KUKA KRL program: Milling_7_2.src

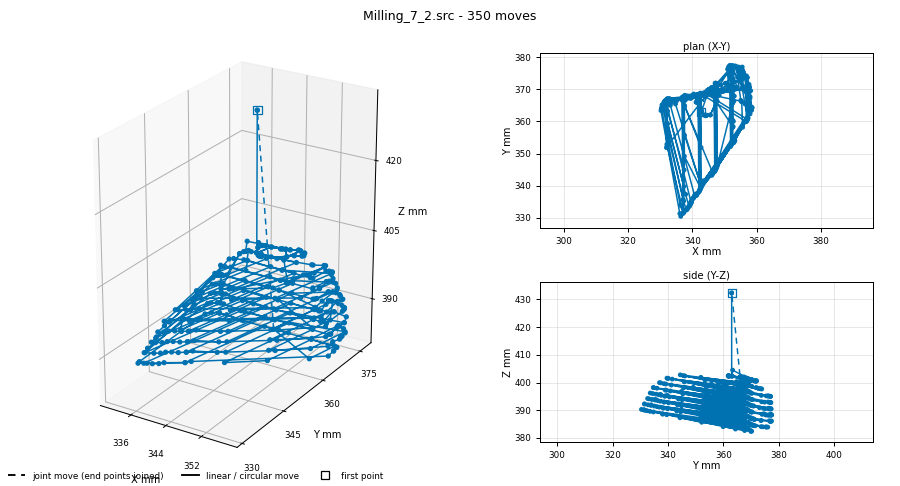
[picture p0: tool path of Milling_7_2.src, 350 of 352 moves have a stored position in this frame; points joined in program order, loops and branches not executed]
&ACCESS RVP
&REL 1
&PARAM TEMPLATE = C:\KRC\Roboter\Template\vorgabe
&PARAM EDITMASK = *
DEF Milling_7_2 ( )


;FOLD INI
;FOLD BASISTECH INI
GLOBAL INTERRUPT DECL 3 WHEN $STOPMESS==TRUE DO IR_STOPM ( )
INTERRUPT ON 3
BAS (#INITMOV,0 )
;ENDFOLD (BASISTECH INI)
;ENDFOLD (INI)

;FOLD STARTPOSITION - BASE IS 0, TOOL IS 5, SPEED IS 15%, POSITION IS A1 5,A2 -90,A3 100,A4 5,A5 -10,A6 -5,E1 0,E2 0,E3 0,E4 0
$BWDSTART = FALSE
PDAT_ACT = {VEL 15,ACC 100,APO_DIST 50}
FDAT_ACT = {TOOL_NO 5,BASE_NO 0,IPO_FRAME #BASE}
BAS (#PTP_PARAMS,15)
PTP  {A1 5,A2 -90,A3 100,A4 5,A5 -10,A6 -5,E1 0,E2 0,E3 0,E4 0}
;ENDFOLD

;FOLD LIN SPEED IS 0.1 m/sec, INTERPOLATION SETTINGS IN FOLD
$VEL.CP=0.1
$ADVANCE=3
;ENDFOLD

BAS(#VEL_PTP,2)
PTP {X 342.707, Y 362.992, Z 432.358, A -116.805, B 80.034, C -131.472, E1 0, E2 0, E3 0, E4 0, S 'B010'}
$VEL.CP=0.012
LIN {X 342.707, Y 362.992, Z 402.358, A -116.805, B 80.034, C -131.472, E1 0, E2 0, E3 0, E4 0}
LIN {X 342.661, Y 368.658, Z 401.473, A -116.805, B 80.034, C -131.472, E1 0, E2 0, E3 0, E4 0}
LIN {X 347.621, Y 371.786, Z 400.589, A -116.805, B 80.034, C -131.472, E1 0, E2 0, E3 0, E4 0}
LIN {X 347.667, Y 366.252, Z 401.453, A -116.805, B 80.034, C -131.472, E1 0, E2 0, E3 0, E4 0}
LIN {X 345.179, Y 369.984, Z 401.065, A -116.805, B 80.034, C -131.472, E1 0, E2 0, E3 0, E4 0}
LIN {X 345.924, Y 370.498, Z 400.926, A -116.805, B 80.034, C -131.472, E1 0, E2 0, E3 0, E4 0}
LIN {X 347.063, Y 371.85, Z 400.623, A -116.805, B 80.034, C -131.472, E1 0, E2 0, E3 0, E4 0}
LIN {X 347.223, Y 371.899, Z 400.603, A -116.805, B 80.034, C -131.472, E1 0, E2 0, E3 0, E4 0}
LIN {X 348.776, Y 371.334, Z 400.569, A -116.805, B 80.034, C -131.472, E1 0, E2 0, E3 0, E4 0}
LIN {X 349.45, Y 369.842, Z 400.749, A -116.805, B 80.034, C -131.472, E1 0, E2 0, E3 0, E4 0}
LIN {X 349.322, Y 369.366, Z 400.834, A -116.805, B 80.034, C -131.472, E1 0, E2 0, E3 0, E4 0}
LIN {X 348.261, Y 368.158, Z 401.107, A -116.805, B 80.034, C -131.472, E1 0, E2 0, E3 0, E4 0}
LIN {X 345.56, Y 361.988, Z 402.289, A -116.805, B 80.034, C -131.472, E1 0, E2 0, E3 0, E4 0}
LIN {X 344.437, Y 361.921, Z 402.389, A -116.805, B 80.034, C -131.472, E1 0, E2 0, E3 0, E4 0}
LIN {X 344.141, Y 361.749, Z 402.439, A -116.805, B 80.034, C -131.472, E1 0, E2 0, E3 0, E4 0}
LIN {X 343.696, Y 361.979, Z 402.438, A -116.805, B 80.034, C -131.472, E1 0, E2 0, E3 0, E4 0}
LIN {X 342.553, Y 363.151, Z 402.345, A -116.805, B 80.034, C -131.472, E1 0, E2 0, E3 0, E4 0}
LIN {X 341.15, Y 365.964, Z 402.015, A -116.805, B 80.034, C -131.472, E1 0, E2 0, E3 0, E4 0}
LIN {X 341.012, Y 367.77, Z 401.743, A -116.805, B 80.034, C -131.472, E1 0, E2 0, E3 0, E4 0}
LIN {X 341.478, Y 368.328, Z 401.618, A -116.805, B 80.034, C -131.472, E1 0, E2 0, E3 0, E4 0}
LIN {X 344.42, Y 369.322, Z 401.229, A -116.805, B 80.034, C -131.472, E1 0, E2 0, E3 0, E4 0}
LIN {X 344.649, Y 369.619, Z 401.165, A -116.805, B 80.034, C -131.472, E1 0, E2 0, E3 0, E4 0}
LIN {X 345.179, Y 369.984, Z 401.065, A -116.805, B 80.034, C -131.472, E1 0, E2 0, E3 0, E4 0}
LIN {X 342.877, Y 363.328, Z 404.499, A -116.805, B 80.034, C -131.472, E1 0, E2 0, E3 0, E4 0}
LIN {X 342.707, Y 362.992, Z 402.358, A -116.805, B 80.034, C -131.472, E1 0, E2 0, E3 0, E4 0}
LIN {X 342.661, Y 368.658, Z 401.473, A -116.805, B 80.034, C -131.472, E1 0, E2 0, E3 0, E4 0}
LIN {X 347.621, Y 371.786, Z 400.589, A -116.805, B 80.034, C -131.472, E1 0, E2 0, E3 0, E4 0}
LIN {X 347.667, Y 366.252, Z 401.453, A -116.805, B 80.034, C -131.472, E1 0, E2 0, E3 0, E4 0}
LIN {X 345.179, Y 369.984, Z 401.065, A -116.805, B 80.034, C -131.472, E1 0, E2 0, E3 0, E4 0}
LIN {X 345.924, Y 370.498, Z 400.926, A -116.805, B 80.034, C -131.472, E1 0, E2 0, E3 0, E4 0}
LIN {X 347.063, Y 371.85, Z 400.623, A -116.805, B 80.034, C -131.472, E1 0, E2 0, E3 0, E4 0}
LIN {X 347.223, Y 371.899, Z 400.603, A -116.805, B 80.034, C -131.472, E1 0, E2 0, E3 0, E4 0}
LIN {X 348.776, Y 371.334, Z 400.569, A -116.805, B 80.034, C -131.472, E1 0, E2 0, E3 0, E4 0}
LIN {X 349.45, Y 369.842, Z 400.749, A -116.805, B 80.034, C -131.472, E1 0, E2 0, E3 0, E4 0}
LIN {X 349.322, Y 369.366, Z 400.834, A -116.805, B 80.034, C -131.472, E1 0, E2 0, E3 0, E4 0}
LIN {X 348.261, Y 368.158, Z 401.107, A -116.805, B 80.034, C -131.472, E1 0, E2 0, E3 0, E4 0}
LIN {X 345.56, Y 361.988, Z 402.289, A -116.805, B 80.034, C -131.472, E1 0, E2 0, E3 0, E4 0}
LIN {X 344.437, Y 361.921, Z 402.389, A -116.805, B 80.034, C -131.472, E1 0, E2 0, E3 0, E4 0}
LIN {X 344.141, Y 361.749, Z 402.439, A -116.805, B 80.034, C -131.472, E1 0, E2 0, E3 0, E4 0}
LIN {X 343.696, Y 361.979, Z 402.438, A -116.805, B 80.034, C -131.472, E1 0, E2 0, E3 0, E4 0}
LIN {X 342.553, Y 363.151, Z 402.345, A -116.805, B 80.034, C -131.472, E1 0, E2 0, E3 0, E4 0}
LIN {X 341.15, Y 365.964, Z 402.015, A -116.805, B 80.034, C -131.472, E1 0, E2 0, E3 0, E4 0}
LIN {X 341.012, Y 367.77, Z 401.743, A -116.805, B 80.034, C -131.472, E1 0, E2 0, E3 0, E4 0}
LIN {X 341.478, Y 368.328, Z 401.618, A -116.805, B 80.034, C -131.472, E1 0, E2 0, E3 0, E4 0}
LIN {X 344.42, Y 369.322, Z 401.229, A -116.805, B 80.034, C -131.472, E1 0, E2 0, E3 0, E4 0}
LIN {X 344.649, Y 369.619, Z 401.165, A -116.805, B 80.034, C -131.472, E1 0, E2 0, E3 0, E4 0}
LIN {X 345.179, Y 369.984, Z 401.065, A -116.805, B 80.034, C -131.472, E1 0, E2 0, E3 0, E4 0}
LIN {X 337.743, Y 367.407, Z 402.059, A -116.805, B 80.034, C -131.472, E1 0, E2 0, E3 0, E4 0}
LIN {X 337.573, Y 367.071, Z 399.918, A -116.805, B 80.034, C -131.472, E1 0, E2 0, E3 0, E4 0}
LIN {X 337.592, Y 364.763, Z 400.278, A -116.805, B 80.034, C -131.472, E1 0, E2 0, E3 0, E4 0}
LIN {X 342.685, Y 351.876, Z 401.896, A -116.805, B 80.034, C -131.472, E1 0, E2 0, E3 0, E4 0}
LIN {X 342.545, Y 368.751, Z 399.26, A -116.805, B 80.034, C -131.472, E1 0, E2 0, E3 0, E4 0}
LIN {X 347.519, Y 370.271, Z 398.628, A -116.805, B 80.034, C -131.472, E1 0, E2 0, E3 0, E4 0}
LIN {X 347.718, Y 346.142, Z 402.396, A -116.805, B 80.034, C -131.472, E1 0, E2 0, E3 0, E4 0}
LIN {X 352.543, Y 365.664, Z 398.952, A -116.805, B 80.034, C -131.472, E1 0, E2 0, E3 0, E4 0}
LIN {X 352.483, Y 372.939, Z 397.816, A -116.805, B 80.034, C -131.472, E1 0, E2 0, E3 0, E4 0}
LIN {X 352.587, Y 360.294, Z 399.791, A -116.805, B 80.034, C -131.472, E1 0, E2 0, E3 0, E4 0}
LIN {X 352.604, Y 358.316, Z 400.1, A -116.805, B 80.034, C -131.472, E1 0, E2 0, E3 0, E4 0}
LIN {X 345.127, Y 369.414, Z 398.952, A -116.805, B 80.034, C -131.472, E1 0, E2 0, E3 0, E4 0}
LIN {X 350.17, Y 371.833, Z 398.173, A -116.805, B 80.034, C -131.472, E1 0, E2 0, E3 0, E4 0}
LIN {X 350.43, Y 371.898, Z 398.142, A -116.805, B 80.034, C -131.472, E1 0, E2 0, E3 0, E4 0}
LIN {X 351.948, Y 373.669, Z 397.744, A -116.805, B 80.034, C -131.472, E1 0, E2 0, E3 0, E4 0}
LIN {X 352.209, Y 373.838, Z 397.697, A -116.805, B 80.034, C -131.472, E1 0, E2 0, E3 0, E4 0}
LIN {X 352.325, Y 373.23, Z 397.783, A -116.805, B 80.034, C -131.472, E1 0, E2 0, E3 0, E4 0}
LIN {X 352.575, Y 372.77, Z 397.835, A -116.805, B 80.034, C -131.472, E1 0, E2 0, E3 0, E4 0}
LIN {X 353.028, Y 367.871, Z 398.567, A -116.805, B 80.034, C -131.472, E1 0, E2 0, E3 0, E4 0}
LIN {X 352.901, Y 366.299, Z 398.824, A -116.805, B 80.034, C -131.472, E1 0, E2 0, E3 0, E4 0}
LIN {X 352.206, Y 365.066, Z 399.072, A -116.805, B 80.034, C -131.472, E1 0, E2 0, E3 0, E4 0}
LIN {X 352.083, Y 361.375, Z 399.661, A -116.805, B 80.034, C -131.472, E1 0, E2 0, E3 0, E4 0}
LIN {X 352.727, Y 359.98, Z 399.829, A -116.805, B 80.034, C -131.472, E1 0, E2 0, E3 0, E4 0}
LIN {X 352.636, Y 358.39, Z 400.085, A -116.805, B 80.034, C -131.472, E1 0, E2 0, E3 0, E4 0}
LIN {X 352.49, Y 358.055, Z 400.15, A -116.805, B 80.034, C -131.472, E1 0, E2 0, E3 0, E4 0}
LIN {X 352.27, Y 353.357, Z 400.904, A -116.805, B 80.034, C -131.472, E1 0, E2 0, E3 0, E4 0}
LIN {X 347.282, Y 345.532, Z 402.526, A -116.805, B 80.034, C -131.472, E1 0, E2 0, E3 0, E4 0}
LIN {X 346.146, Y 344.436, Z 402.788, A -116.805, B 80.034, C -131.472, E1 0, E2 0, E3 0, E4 0}
LIN {X 337.557, Y 364.832, Z 400.27, A -116.805, B 80.034, C -131.472, E1 0, E2 0, E3 0, E4 0}
LIN {X 337.427, Y 366.588, Z 400.005, A -116.805, B 80.034, C -131.472, E1 0, E2 0, E3 0, E4 0}
LIN {X 337.628, Y 367.255, Z 399.884, A -116.805, B 80.034, C -131.472, E1 0, E2 0, E3 0, E4 0}
LIN {X 338.367, Y 367.942, Z 399.718, A -116.805, B 80.034, C -131.472, E1 0, E2 0, E3 0, E4 0}
LIN {X 340.366, Y 368.526, Z 399.468, A -116.805, B 80.034, C -131.472, E1 0, E2 0, E3 0, E4 0}
LIN {X 343.878, Y 368.815, Z 399.145, A -116.805, B 80.034, C -131.472, E1 0, E2 0, E3 0, E4 0}
LIN {X 345.127, Y 369.414, Z 398.952, A -116.805, B 80.034, C -131.472, E1 0, E2 0, E3 0, E4 0}
LIN {X 337.622, Y 368.124, Z 399.749, A -116.805, B 80.034, C -131.472, E1 0, E2 0, E3 0, E4 0}
LIN {X 337.452, Y 367.788, Z 397.607, A -116.805, B 80.034, C -131.472, E1 0, E2 0, E3 0, E4 0}
LIN {X 337.553, Y 355.652, Z 399.503, A -116.805, B 80.034, C -131.472, E1 0, E2 0, E3 0, E4 0}
LIN {X 342.668, Y 340.052, Z 401.544, A -116.805, B 80.034, C -131.472, E1 0, E2 0, E3 0, E4 0}
LIN {X 342.43, Y 368.782, Z 397.057, A -116.805, B 80.034, C -131.472, E1 0, E2 0, E3 0, E4 0}
LIN {X 347.41, Y 369.598, Z 396.535, A -116.805, B 80.034, C -131.472, E1 0, E2 0, E3 0, E4 0}
LIN {X 347.606, Y 345.887, Z 400.238, A -116.805, B 80.034, C -131.472, E1 0, E2 0, E3 0, E4 0}
LIN {X 352.527, Y 353.746, Z 398.615, A -116.805, B 80.034, C -131.472, E1 0, E2 0, E3 0, E4 0}
LIN {X 352.342, Y 376.171, Z 395.113, A -116.805, B 80.034, C -131.472, E1 0, E2 0, E3 0, E4 0}
LIN {X 344.968, Y 369.019, Z 396.819, A -116.805, B 80.034, C -131.472, E1 0, E2 0, E3 0, E4 0}
LIN {X 350.898, Y 370.064, Z 396.185, A -116.805, B 80.034, C -131.472, E1 0, E2 0, E3 0, E4 0}
LIN {X 351.378, Y 370.235, Z 396.12, A -116.805, B 80.034, C -131.472, E1 0, E2 0, E3 0, E4 0}
LIN {X 350.95, Y 376.236, Z 395.213, A -116.805, B 80.034, C -131.472, E1 0, E2 0, E3 0, E4 0}
LIN {X 351.301, Y 376.912, Z 395.079, A -116.805, B 80.034, C -131.472, E1 0, E2 0, E3 0, E4 0}
LIN {X 351.971, Y 377.016, Z 395.01, A -116.805, B 80.034, C -131.472, E1 0, E2 0, E3 0, E4 0}
LIN {X 352.014, Y 376.959, Z 395.015, A -116.805, B 80.034, C -131.472, E1 0, E2 0, E3 0, E4 0}
LIN {X 352.596, Y 375.492, Z 395.199, A -116.805, B 80.034, C -131.472, E1 0, E2 0, E3 0, E4 0}
LIN {X 354.046, Y 373.693, Z 395.366, A -116.805, B 80.034, C -131.472, E1 0, E2 0, E3 0, E4 0}
LIN {X 355.039, Y 366.561, Z 396.406, A -116.805, B 80.034, C -131.472, E1 0, E2 0, E3 0, E4 0}
LIN {X 355.162, Y 366.239, Z 396.447, A -116.805, B 80.034, C -131.472, E1 0, E2 0, E3 0, E4 0}
LIN {X 355.322, Y 366.123, Z 396.453, A -116.805, B 80.034, C -131.472, E1 0, E2 0, E3 0, E4 0}
LIN {X 355.617, Y 358.157, Z 397.679, A -116.805, B 80.034, C -131.472, E1 0, E2 0, E3 0, E4 0}
LIN {X 343.462, Y 341.535, Z 401.249, A -116.805, B 80.034, C -131.472, E1 0, E2 0, E3 0, E4 0}
LIN {X 342.983, Y 340.017, Z 401.525, A -116.805, B 80.034, C -131.472, E1 0, E2 0, E3 0, E4 0}
LIN {X 342.757, Y 339.627, Z 401.604, A -116.805, B 80.034, C -131.472, E1 0, E2 0, E3 0, E4 0}
LIN {X 334.72, Y 365.41, Z 398.197, A -116.805, B 80.034, C -131.472, E1 0, E2 0, E3 0, E4 0}
LIN {X 335.142, Y 366.46, Z 397.999, A -116.805, B 80.034, C -131.472, E1 0, E2 0, E3 0, E4 0}
LIN {X 336.836, Y 367.584, Z 397.688, A -116.805, B 80.034, C -131.472, E1 0, E2 0, E3 0, E4 0}
LIN {X 344.968, Y 369.019, Z 396.819, A -116.805, B 80.034, C -131.472, E1 0, E2 0, E3 0, E4 0}
LIN {X 337.509, Y 367.931, Z 397.58, A -116.805, B 80.034, C -131.472, E1 0, E2 0, E3 0, E4 0}
LIN {X 337.339, Y 367.595, Z 395.439, A -116.805, B 80.034, C -131.472, E1 0, E2 0, E3 0, E4 0}
LIN {X 337.492, Y 349.128, Z 398.324, A -116.805, B 80.034, C -131.472, E1 0, E2 0, E3 0, E4 0}
LIN {X 342.56, Y 339.244, Z 399.472, A -116.805, B 80.034, C -131.472, E1 0, E2 0, E3 0, E4 0}
LIN {X 342.317, Y 368.636, Z 394.882, A -116.805, B 80.034, C -131.472, E1 0, E2 0, E3 0, E4 0}
LIN {X 347.298, Y 369.262, Z 394.389, A -116.805, B 80.034, C -131.472, E1 0, E2 0, E3 0, E4 0}
LIN {X 347.493, Y 345.631, Z 398.08, A -116.805, B 80.034, C -131.472, E1 0, E2 0, E3 0, E4 0}
LIN {X 352.414, Y 353.489, Z 396.457, A -116.805, B 80.034, C -131.472, E1 0, E2 0, E3 0, E4 0}
LIN {X 352.22, Y 377.058, Z 392.776, A -116.805, B 80.034, C -131.472, E1 0, E2 0, E3 0, E4 0}
LIN {X 344.8, Y 368.674, Z 394.679, A -116.805, B 80.034, C -131.472, E1 0, E2 0, E3 0, E4 0}
LIN {X 351.511, Y 369.969, Z 393.944, A -116.805, B 80.034, C -131.472, E1 0, E2 0, E3 0, E4 0}
LIN {X 351.273, Y 370.494, Z 393.881, A -116.805, B 80.034, C -131.472, E1 0, E2 0, E3 0, E4 0}
LIN {X 351.117, Y 376.143, Z 393.007, A -116.805, B 80.034, C -131.472, E1 0, E2 0, E3 0, E4 0}
LIN {X 351.368, Y 376.885, Z 392.871, A -116.805, B 80.034, C -131.472, E1 0, E2 0, E3 0, E4 0}
LIN {X 351.939, Y 377.152, Z 392.784, A -116.805, B 80.034, C -131.472, E1 0, E2 0, E3 0, E4 0}
LIN {X 352.88, Y 376.879, Z 392.752, A -116.805, B 80.034, C -131.472, E1 0, E2 0, E3 0, E4 0}
LIN {X 354.436, Y 374.837, Z 392.949, A -116.805, B 80.034, C -131.472, E1 0, E2 0, E3 0, E4 0}
LIN {X 354.922, Y 373.812, Z 393.071, A -116.805, B 80.034, C -131.472, E1 0, E2 0, E3 0, E4 0}
LIN {X 356.33, Y 365.429, Z 394.274, A -116.805, B 80.034, C -131.472, E1 0, E2 0, E3 0, E4 0}
LIN {X 357.254, Y 361.21, Z 394.863, A -116.805, B 80.034, C -131.472, E1 0, E2 0, E3 0, E4 0}
LIN {X 357.256, Y 360.934, Z 394.906, A -116.805, B 80.034, C -131.472, E1 0, E2 0, E3 0, E4 0}
LIN {X 343.292, Y 341.2, Z 399.108, A -116.805, B 80.034, C -131.472, E1 0, E2 0, E3 0, E4 0}
LIN {X 342.161, Y 338.545, Z 399.614, A -116.805, B 80.034, C -131.472, E1 0, E2 0, E3 0, E4 0}
LIN {X 340.955, Y 337.378, Z 399.892, A -116.805, B 80.034, C -131.472, E1 0, E2 0, E3 0, E4 0}
LIN {X 340.651, Y 336.946, Z 399.984, A -116.805, B 80.034, C -131.472, E1 0, E2 0, E3 0, E4 0}
LIN {X 333.128, Y 365.005, Z 396.179, A -116.805, B 80.034, C -131.472, E1 0, E2 0, E3 0, E4 0}
LIN {X 333.456, Y 365.891, Z 396.015, A -116.805, B 80.034, C -131.472, E1 0, E2 0, E3 0, E4 0}
LIN {X 334.317, Y 366.652, Z 395.827, A -116.805, B 80.034, C -131.472, E1 0, E2 0, E3 0, E4 0}
LIN {X 344.8, Y 368.674, Z 394.679, A -116.805, B 80.034, C -131.472, E1 0, E2 0, E3 0, E4 0}
LIN {X 332.426, Y 365.828, Z 396.106, A -116.805, B 80.034, C -131.472, E1 0, E2 0, E3 0, E4 0}
LIN {X 332.256, Y 365.492, Z 393.965, A -116.805, B 80.034, C -131.472, E1 0, E2 0, E3 0, E4 0}
LIN {X 332.275, Y 363.181, Z 394.326, A -116.805, B 80.034, C -131.472, E1 0, E2 0, E3 0, E4 0}
LIN {X 337.412, Y 344.878, Z 396.789, A -116.805, B 80.034, C -131.472, E1 0, E2 0, E3 0, E4 0}
LIN {X 337.226, Y 367.425, Z 393.268, A -116.805, B 80.034, C -131.472, E1 0, E2 0, E3 0, E4 0}
LIN {X 342.205, Y 368.272, Z 392.74, A -116.805, B 80.034, C -131.472, E1 0, E2 0, E3 0, E4 0}
LIN {X 342.447, Y 339.008, Z 397.311, A -116.805, B 80.034, C -131.472, E1 0, E2 0, E3 0, E4 0}
LIN {X 347.381, Y 345.375, Z 395.921, A -116.805, B 80.034, C -131.472, E1 0, E2 0, E3 0, E4 0}
LIN {X 347.184, Y 369.21, Z 392.199, A -116.805, B 80.034, C -131.472, E1 0, E2 0, E3 0, E4 0}
LIN {X 352.105, Y 377.077, Z 390.575, A -116.805, B 80.034, C -131.472, E1 0, E2 0, E3 0, E4 0}
LIN {X 352.302, Y 353.231, Z 394.299, A -116.805, B 80.034, C -131.472, E1 0, E2 0, E3 0, E4 0}
LIN {X 357.225, Y 360.845, Z 392.715, A -116.805, B 80.034, C -131.472, E1 0, E2 0, E3 0, E4 0}
LIN {X 357.184, Y 365.844, Z 391.934, A -116.805, B 80.034, C -131.472, E1 0, E2 0, E3 0, E4 0}
LIN {X 344.593, Y 368.511, Z 392.514, A -116.805, B 80.034, C -131.472, E1 0, E2 0, E3 0, E4 0}
LIN {X 351.639, Y 369.951, Z 391.73, A -116.805, B 80.034, C -131.472, E1 0, E2 0, E3 0, E4 0}
LIN {X 351.935, Y 370.164, Z 391.673, A -116.805, B 80.034, C -131.472, E1 0, E2 0, E3 0, E4 0}
LIN {X 351.921, Y 370.773, Z 391.578, A -116.805, B 80.034, C -131.472, E1 0, E2 0, E3 0, E4 0}
LIN {X 351.982, Y 370.93, Z 391.549, A -116.805, B 80.034, C -131.472, E1 0, E2 0, E3 0, E4 0}
LIN {X 351.507, Y 376.272, Z 390.749, A -116.805, B 80.034, C -131.472, E1 0, E2 0, E3 0, E4 0}
LIN {X 351.55, Y 376.484, Z 390.712, A -116.805, B 80.034, C -131.472, E1 0, E2 0, E3 0, E4 0}
LIN {X 352.162, Y 377.157, Z 390.558, A -116.805, B 80.034, C -131.472, E1 0, E2 0, E3 0, E4 0}
LIN {X 352.82, Y 377.236, Z 390.493, A -116.805, B 80.034, C -131.472, E1 0, E2 0, E3 0, E4 0}
LIN {X 353.837, Y 376.969, Z 390.455, A -116.805, B 80.034, C -131.472, E1 0, E2 0, E3 0, E4 0}
LIN {X 354.308, Y 376.387, Z 390.509, A -116.805, B 80.034, C -131.472, E1 0, E2 0, E3 0, E4 0}
LIN {X 355.568, Y 375.15, Z 390.603, A -116.805, B 80.034, C -131.472, E1 0, E2 0, E3 0, E4 0}
LIN {X 355.65, Y 374.457, Z 390.705, A -116.805, B 80.034, C -131.472, E1 0, E2 0, E3 0, E4 0}
LIN {X 355.5, Y 373.025, Z 390.942, A -116.805, B 80.034, C -131.472, E1 0, E2 0, E3 0, E4 0}
LIN {X 357.931, Y 362.32, Z 392.428, A -116.805, B 80.034, C -131.472, E1 0, E2 0, E3 0, E4 0}
LIN {X 343.123, Y 340.864, Z 396.966, A -116.805, B 80.034, C -131.472, E1 0, E2 0, E3 0, E4 0}
LIN {X 342.665, Y 339.388, Z 397.234, A -116.805, B 80.034, C -131.472, E1 0, E2 0, E3 0, E4 0}
LIN {X 340.081, Y 336.066, Z 397.96, A -116.805, B 80.034, C -131.472, E1 0, E2 0, E3 0, E4 0}
LIN {X 339.703, Y 334.863, Z 398.179, A -116.805, B 80.034, C -131.472, E1 0, E2 0, E3 0, E4 0}
LIN {X 339.587, Y 334.711, Z 398.212, A -116.805, B 80.034, C -131.472, E1 0, E2 0, E3 0, E4 0}
LIN {X 332.028, Y 364.986, Z 394.062, A -116.805, B 80.034, C -131.472, E1 0, E2 0, E3 0, E4 0}
LIN {X 332.055, Y 365.12, Z 394.039, A -116.805, B 80.034, C -131.472, E1 0, E2 0, E3 0, E4 0}
LIN {X 332.306, Y 365.585, Z 393.946, A -116.805, B 80.034, C -131.472, E1 0, E2 0, E3 0, E4 0}
LIN {X 332.861, Y 366.112, Z 393.82, A -116.805, B 80.034, C -131.472, E1 0, E2 0, E3 0, E4 0}
LIN {X 344.593, Y 368.511, Z 392.514, A -116.805, B 80.034, C -131.472, E1 0, E2 0, E3 0, E4 0}
LIN {X 332.306, Y 366.393, Z 393.82, A -116.805, B 80.034, C -131.472, E1 0, E2 0, E3 0, E4 0}
LIN {X 332.137, Y 366.057, Z 391.678, A -116.805, B 80.034, C -131.472, E1 0, E2 0, E3 0, E4 0}
LIN {X 332.193, Y 359.284, Z 392.736, A -116.805, B 80.034, C -131.472, E1 0, E2 0, E3 0, E4 0}
LIN {X 332.193, Y 359.252, Z 392.741, A -116.805, B 80.034, C -131.472, E1 0, E2 0, E3 0, E4 0}
LIN {X 337.34, Y 339.742, Z 395.393, A -116.805, B 80.034, C -131.472, E1 0, E2 0, E3 0, E4 0}
LIN {X 337.115, Y 367.064, Z 391.126, A -116.805, B 80.034, C -131.472, E1 0, E2 0, E3 0, E4 0}
LIN {X 342.095, Y 367.705, Z 390.631, A -116.805, B 80.034, C -131.472, E1 0, E2 0, E3 0, E4 0}
LIN {X 342.334, Y 338.772, Z 395.15, A -116.805, B 80.034, C -131.472, E1 0, E2 0, E3 0, E4 0}
LIN {X 347.268, Y 345.12, Z 393.763, A -116.805, B 80.034, C -131.472, E1 0, E2 0, E3 0, E4 0}
LIN {X 347.07, Y 369.058, Z 390.024, A -116.805, B 80.034, C -131.472, E1 0, E2 0, E3 0, E4 0}
LIN {X 352.049, Y 369.948, Z 389.49, A -116.805, B 80.034, C -131.472, E1 0, E2 0, E3 0, E4 0}
LIN {X 352.19, Y 352.974, Z 392.141, A -116.805, B 80.034, C -131.472, E1 0, E2 0, E3 0, E4 0}
LIN {X 352.011, Y 374.625, Z 388.76, A -116.805, B 80.034, C -131.472, E1 0, E2 0, E3 0, E4 0}
LIN {X 351.988, Y 377.367, Z 388.332, A -116.805, B 80.034, C -131.472, E1 0, E2 0, E3 0, E4 0}
LIN {X 357.056, Y 367.496, Z 389.478, A -116.805, B 80.034, C -131.472, E1 0, E2 0, E3 0, E4 0}
LIN {X 357.113, Y 360.611, Z 390.553, A -116.805, B 80.034, C -131.472, E1 0, E2 0, E3 0, E4 0}
LIN {X 344.36, Y 368.499, Z 390.327, A -116.805, B 80.034, C -131.472, E1 0, E2 0, E3 0, E4 0}
LIN {X 332.559, Y 366.382, Z 391.594, A -116.805, B 80.034, C -131.472, E1 0, E2 0, E3 0, E4 0}
LIN {X 331.405, Y 365.485, Z 391.826, A -116.805, B 80.034, C -131.472, E1 0, E2 0, E3 0, E4 0}
LIN {X 331.047, Y 364.758, Z 391.969, A -116.805, B 80.034, C -131.472, E1 0, E2 0, E3 0, E4 0}
LIN {X 337.873, Y 337.305, Z 395.733, A -116.805, B 80.034, C -131.472, E1 0, E2 0, E3 0, E4 0}
LIN {X 338.86, Y 333.599, Z 396.236, A -116.805, B 80.034, C -131.472, E1 0, E2 0, E3 0, E4 0}
LIN {X 339.534, Y 334.527, Z 396.037, A -116.805, B 80.034, C -131.472, E1 0, E2 0, E3 0, E4 0}
LIN {X 339.911, Y 335.73, Z 395.819, A -116.805, B 80.034, C -131.472, E1 0, E2 0, E3 0, E4 0}
LIN {X 340.616, Y 336.707, Z 395.61, A -116.805, B 80.034, C -131.472, E1 0, E2 0, E3 0, E4 0}
LIN {X 341.575, Y 337.565, Z 395.399, A -116.805, B 80.034, C -131.472, E1 0, E2 0, E3 0, E4 0}
LIN {X 342.474, Y 339.01, Z 395.101, A -116.805, B 80.034, C -131.472, E1 0, E2 0, E3 0, E4 0}
LIN {X 342.953, Y 340.528, Z 394.825, A -116.805, B 80.034, C -131.472, E1 0, E2 0, E3 0, E4 0}
LIN {X 346.357, Y 343.857, Z 394.033, A -116.805, B 80.034, C -131.472, E1 0, E2 0, E3 0, E4 0}
LIN {X 353.213, Y 354.048, Z 391.892, A -116.805, B 80.034, C -131.472, E1 0, E2 0, E3 0, E4 0}
LIN {X 358.337, Y 363.399, Z 390.019, A -116.805, B 80.034, C -131.472, E1 0, E2 0, E3 0, E4 0}
LIN {X 357.551, Y 365.124, Z 389.811, A -116.805, B 80.034, C -131.472, E1 0, E2 0, E3 0, E4 0}
LIN {X 356.182, Y 373.976, Z 388.531, A -116.805, B 80.034, C -131.472, E1 0, E2 0, E3 0, E4 0}
LIN {X 355.88, Y 375.192, Z 388.364, A -116.805, B 80.034, C -131.472, E1 0, E2 0, E3 0, E4 0}
LIN {X 355.724, Y 375.409, Z 388.343, A -116.805, B 80.034, C -131.472, E1 0, E2 0, E3 0, E4 0}
LIN {X 355.54, Y 375.992, Z 388.266, A -116.805, B 80.034, C -131.472, E1 0, E2 0, E3 0, E4 0}
LIN {X 355.366, Y 376.235, Z 388.242, A -116.805, B 80.034, C -131.472, E1 0, E2 0, E3 0, E4 0}
LIN {X 354.401, Y 376.91, Z 388.212, A -116.805, B 80.034, C -131.472, E1 0, E2 0, E3 0, E4 0}
LIN {X 353.339, Y 377.254, Z 388.242, A -116.805, B 80.034, C -131.472, E1 0, E2 0, E3 0, E4 0}
LIN {X 351.667, Y 377.381, Z 388.355, A -116.805, B 80.034, C -131.472, E1 0, E2 0, E3 0, E4 0}
LIN {X 351.574, Y 377.331, Z 388.37, A -116.805, B 80.034, C -131.472, E1 0, E2 0, E3 0, E4 0}
LIN {X 351.315, Y 376.949, Z 388.451, A -116.805, B 80.034, C -131.472, E1 0, E2 0, E3 0, E4 0}
LIN {X 351.3, Y 376.862, Z 388.466, A -116.805, B 80.034, C -131.472, E1 0, E2 0, E3 0, E4 0}
LIN {X 353.236, Y 370.362, Z 389.331, A -116.805, B 80.034, C -131.472, E1 0, E2 0, E3 0, E4 0}
LIN {X 352.984, Y 370.157, Z 389.383, A -116.805, B 80.034, C -131.472, E1 0, E2 0, E3 0, E4 0}
LIN {X 352.945, Y 370.038, Z 389.405, A -116.805, B 80.034, C -131.472, E1 0, E2 0, E3 0, E4 0}
LIN {X 344.36, Y 368.499, Z 390.327, A -116.805, B 80.034, C -131.472, E1 0, E2 0, E3 0, E4 0}
LIN {X 332.186, Y 367.091, Z 391.512, A -116.805, B 80.034, C -131.472, E1 0, E2 0, E3 0, E4 0}
LIN {X 332.016, Y 366.755, Z 389.371, A -116.805, B 80.034, C -131.472, E1 0, E2 0, E3 0, E4 0}
LIN {X 332.1, Y 356.639, Z 390.951, A -116.805, B 80.034, C -131.472, E1 0, E2 0, E3 0, E4 0}
LIN {X 337.263, Y 335.2, Z 393.905, A -116.805, B 80.034, C -131.472, E1 0, E2 0, E3 0, E4 0}
LIN {X 337.002, Y 366.813, Z 388.967, A -116.805, B 80.034, C -131.472, E1 0, E2 0, E3 0, E4 0}
LIN {X 341.982, Y 367.627, Z 388.445, A -116.805, B 80.034, C -131.472, E1 0, E2 0, E3 0, E4 0}
LIN {X 342.222, Y 338.536, Z 392.989, A -116.805, B 80.034, C -131.472, E1 0, E2 0, E3 0, E4 0}
LIN {X 347.156, Y 344.864, Z 391.605, A -116.805, B 80.034, C -131.472, E1 0, E2 0, E3 0, E4 0}
LIN {X 346.957, Y 368.945, Z 387.844, A -116.805, B 80.034, C -131.472, E1 0, E2 0, E3 0, E4 0}
LIN {X 351.936, Y 369.823, Z 387.312, A -116.805, B 80.034, C -131.472, E1 0, E2 0, E3 0, E4 0}
LIN {X 352.077, Y 352.728, Z 389.982, A -116.805, B 80.034, C -131.472, E1 0, E2 0, E3 0, E4 0}
LIN {X 352.077, Y 352.716, Z 389.984, A -116.805, B 80.034, C -131.472, E1 0, E2 0, E3 0, E4 0}
LIN {X 357, Y 360.377, Z 388.392, A -116.805, B 80.034, C -131.472, E1 0, E2 0, E3 0, E4 0}
LIN {X 356.915, Y 371.134, Z 386.712, A -116.805, B 80.034, C -131.472, E1 0, E2 0, E3 0, E4 0}
LIN {X 356.911, Y 371.19, Z 386.703, A -116.805, B 80.034, C -131.472, E1 0, E2 0, E3 0, E4 0}
LIN {X 356.891, Y 373.563, Z 386.332, A -116.805, B 80.034, C -131.472, E1 0, E2 0, E3 0, E4 0}
LIN {X 344.2, Y 368.122, Z 388.191, A -116.805, B 80.034, C -131.472, E1 0, E2 0, E3 0, E4 0}
LIN {X 339.425, Y 367.119, Z 388.727, A -116.805, B 80.034, C -131.472, E1 0, E2 0, E3 0, E4 0}
LIN {X 332.76, Y 367.131, Z 389.253, A -116.805, B 80.034, C -131.472, E1 0, E2 0, E3 0, E4 0}
LIN {X 331.843, Y 366.668, Z 389.399, A -116.805, B 80.034, C -131.472, E1 0, E2 0, E3 0, E4 0}
LIN {X 331.043, Y 365.812, Z 389.596, A -116.805, B 80.034, C -131.472, E1 0, E2 0, E3 0, E4 0}
LIN {X 330.639, Y 364.816, Z 389.785, A -116.805, B 80.034, C -131.472, E1 0, E2 0, E3 0, E4 0}
LIN {X 337.082, Y 335.728, Z 393.836, A -116.805, B 80.034, C -131.472, E1 0, E2 0, E3 0, E4 0}
LIN {X 337.989, Y 332.648, Z 394.247, A -116.805, B 80.034, C -131.472, E1 0, E2 0, E3 0, E4 0}
LIN {X 338.595, Y 333.131, Z 394.124, A -116.805, B 80.034, C -131.472, E1 0, E2 0, E3 0, E4 0}
LIN {X 339.364, Y 334.191, Z 393.896, A -116.805, B 80.034, C -131.472, E1 0, E2 0, E3 0, E4 0}
LIN {X 339.741, Y 335.394, Z 393.678, A -116.805, B 80.034, C -131.472, E1 0, E2 0, E3 0, E4 0}
LIN {X 340.446, Y 336.371, Z 393.469, A -116.805, B 80.034, C -131.472, E1 0, E2 0, E3 0, E4 0}
LIN {X 341.406, Y 337.229, Z 393.258, A -116.805, B 80.034, C -131.472, E1 0, E2 0, E3 0, E4 0}
LIN {X 342.305, Y 338.674, Z 392.96, A -116.805, B 80.034, C -131.472, E1 0, E2 0, E3 0, E4 0}
LIN {X 342.784, Y 340.193, Z 392.684, A -116.805, B 80.034, C -131.472, E1 0, E2 0, E3 0, E4 0}
LIN {X 346.187, Y 343.521, Z 391.892, A -116.805, B 80.034, C -131.472, E1 0, E2 0, E3 0, E4 0}
LIN {X 353.044, Y 353.713, Z 389.751, A -116.805, B 80.034, C -131.472, E1 0, E2 0, E3 0, E4 0}
LIN {X 358.354, Y 363.527, Z 387.791, A -116.805, B 80.034, C -131.472, E1 0, E2 0, E3 0, E4 0}
LIN {X 357.272, Y 369.957, Z 386.868, A -116.805, B 80.034, C -131.472, E1 0, E2 0, E3 0, E4 0}
LIN {X 356.915, Y 371.134, Z 386.712, A -116.805, B 80.034, C -131.472, E1 0, E2 0, E3 0, E4 0}
LIN {X 356.886, Y 373.607, Z 386.326, A -116.805, B 80.034, C -131.472, E1 0, E2 0, E3 0, E4 0}
LIN {X 355.486, Y 376.921, Z 385.917, A -116.805, B 80.034, C -131.472, E1 0, E2 0, E3 0, E4 0}
LIN {X 352.435, Y 377.319, Z 386.096, A -116.805, B 80.034, C -131.472, E1 0, E2 0, E3 0, E4 0}
LIN {X 352.403, Y 377.305, Z 386.101, A -116.805, B 80.034, C -131.472, E1 0, E2 0, E3 0, E4 0}
LIN {X 352.149, Y 376.601, Z 386.232, A -116.805, B 80.034, C -131.472, E1 0, E2 0, E3 0, E4 0}
LIN {X 353.806, Y 370.705, Z 387.025, A -116.805, B 80.034, C -131.472, E1 0, E2 0, E3 0, E4 0}
LIN {X 353.384, Y 370.052, Z 387.161, A -116.805, B 80.034, C -131.472, E1 0, E2 0, E3 0, E4 0}
LIN {X 344.2, Y 368.122, Z 388.191, A -116.805, B 80.034, C -131.472, E1 0, E2 0, E3 0, E4 0}
LIN {X 332.073, Y 366.924, Z 389.341, A -116.805, B 80.034, C -131.472, E1 0, E2 0, E3 0, E4 0}
LIN {X 331.903, Y 366.588, Z 387.199, A -116.805, B 80.034, C -131.472, E1 0, E2 0, E3 0, E4 0}
LIN {X 332.017, Y 352.837, Z 389.347, A -116.805, B 80.034, C -131.472, E1 0, E2 0, E3 0, E4 0}
LIN {X 337.178, Y 331.593, Z 392.27, A -116.805, B 80.034, C -131.472, E1 0, E2 0, E3 0, E4 0}
LIN {X 336.891, Y 366.439, Z 386.827, A -116.805, B 80.034, C -131.472, E1 0, E2 0, E3 0, E4 0}
LIN {X 341.867, Y 367.658, Z 386.242, A -116.805, B 80.034, C -131.472, E1 0, E2 0, E3 0, E4 0}
LIN {X 342.109, Y 338.3, Z 390.827, A -116.805, B 80.034, C -131.472, E1 0, E2 0, E3 0, E4 0}
LIN {X 347.043, Y 344.608, Z 389.447, A -116.805, B 80.034, C -131.472, E1 0, E2 0, E3 0, E4 0}
LIN {X 346.843, Y 368.818, Z 385.666, A -116.805, B 80.034, C -131.472, E1 0, E2 0, E3 0, E4 0}
LIN {X 351.823, Y 369.657, Z 385.139, A -116.805, B 80.034, C -131.472, E1 0, E2 0, E3 0, E4 0}
LIN {X 351.965, Y 352.442, Z 387.828, A -116.805, B 80.034, C -131.472, E1 0, E2 0, E3 0, E4 0}
LIN {X 356.887, Y 360.142, Z 386.23, A -116.805, B 80.034, C -131.472, E1 0, E2 0, E3 0, E4 0}
LIN {X 356.771, Y 374.199, Z 384.035, A -116.805, B 80.034, C -131.472, E1 0, E2 0, E3 0, E4 0}
LIN {X 344.023, Y 367.819, Z 386.046, A -116.805, B 80.034, C -131.472, E1 0, E2 0, E3 0, E4 0}
LIN {X 337.723, Y 366.543, Z 386.745, A -116.805, B 80.034, C -131.472, E1 0, E2 0, E3 0, E4 0}
LIN {X 332.535, Y 366.756, Z 387.123, A -116.805, B 80.034, C -131.472, E1 0, E2 0, E3 0, E4 0}
LIN {X 331.471, Y 366.407, Z 387.262, A -116.805, B 80.034, C -131.472, E1 0, E2 0, E3 0, E4 0}
LIN {X 331.313, Y 366.269, Z 387.296, A -116.805, B 80.034, C -131.472, E1 0, E2 0, E3 0, E4 0}
LIN {X 330.508, Y 365.022, Z 387.556, A -116.805, B 80.034, C -131.472, E1 0, E2 0, E3 0, E4 0}
LIN {X 330.325, Y 364.142, Z 387.708, A -116.805, B 80.034, C -131.472, E1 0, E2 0, E3 0, E4 0}
LIN {X 336.216, Y 333.888, Z 391.986, A -116.805, B 80.034, C -131.472, E1 0, E2 0, E3 0, E4 0}
LIN {X 337.091, Y 331.485, Z 392.294, A -116.805, B 80.034, C -131.472, E1 0, E2 0, E3 0, E4 0}
LIN {X 338.426, Y 332.795, Z 391.983, A -116.805, B 80.034, C -131.472, E1 0, E2 0, E3 0, E4 0}
LIN {X 339.194, Y 333.855, Z 391.755, A -116.805, B 80.034, C -131.472, E1 0, E2 0, E3 0, E4 0}
LIN {X 339.572, Y 335.058, Z 391.537, A -116.805, B 80.034, C -131.472, E1 0, E2 0, E3 0, E4 0}
LIN {X 340.277, Y 336.035, Z 391.328, A -116.805, B 80.034, C -131.472, E1 0, E2 0, E3 0, E4 0}
LIN {X 341.236, Y 336.893, Z 391.117, A -116.805, B 80.034, C -131.472, E1 0, E2 0, E3 0, E4 0}
LIN {X 342.135, Y 338.338, Z 390.819, A -116.805, B 80.034, C -131.472, E1 0, E2 0, E3 0, E4 0}
LIN {X 342.614, Y 339.857, Z 390.543, A -116.805, B 80.034, C -131.472, E1 0, E2 0, E3 0, E4 0}
LIN {X 346.018, Y 343.185, Z 389.751, A -116.805, B 80.034, C -131.472, E1 0, E2 0, E3 0, E4 0}
LIN {X 352.874, Y 353.377, Z 387.61, A -116.805, B 80.034, C -131.472, E1 0, E2 0, E3 0, E4 0}
LIN {X 358.543, Y 364.199, Z 385.463, A -116.805, B 80.034, C -131.472, E1 0, E2 0, E3 0, E4 0}
LIN {X 357.903, Y 367.189, Z 385.045, A -116.805, B 80.034, C -131.472, E1 0, E2 0, E3 0, E4 0}
LIN {X 358.126, Y 369.542, Z 384.658, A -116.805, B 80.034, C -131.472, E1 0, E2 0, E3 0, E4 0}
LIN {X 357.796, Y 370.633, Z 384.513, A -116.805, B 80.034, C -131.472, E1 0, E2 0, E3 0, E4 0}
LIN {X 357.547, Y 370.98, Z 384.478, A -116.805, B 80.034, C -131.472, E1 0, E2 0, E3 0, E4 0}
LIN {X 357.619, Y 371.491, Z 384.393, A -116.805, B 80.034, C -131.472, E1 0, E2 0, E3 0, E4 0}
LIN {X 357.116, Y 373.631, Z 384.097, A -116.805, B 80.034, C -131.472, E1 0, E2 0, E3 0, E4 0}
LIN {X 355.729, Y 375.427, Z 383.925, A -116.805, B 80.034, C -131.472, E1 0, E2 0, E3 0, E4 0}
LIN {X 354.509, Y 376.035, Z 383.926, A -116.805, B 80.034, C -131.472, E1 0, E2 0, E3 0, E4 0}
LIN {X 354.266, Y 375.45, Z 384.037, A -116.805, B 80.034, C -131.472, E1 0, E2 0, E3 0, E4 0}
LIN {X 355.548, Y 370.549, Z 384.704, A -116.805, B 80.034, C -131.472, E1 0, E2 0, E3 0, E4 0}
LIN {X 355.503, Y 370.32, Z 384.744, A -116.805, B 80.034, C -131.472, E1 0, E2 0, E3 0, E4 0}
LIN {X 355.392, Y 370.121, Z 384.784, A -116.805, B 80.034, C -131.472, E1 0, E2 0, E3 0, E4 0}
LIN {X 344.023, Y 367.819, Z 386.046, A -116.805, B 80.034, C -131.472, E1 0, E2 0, E3 0, E4 0}
LIN {X 332.08, Y 352.16, Z 389.448, A -116.805, B 80.034, C -131.472, E1 0, E2 0, E3 0, E4 0}
LIN {X 331.91, Y 351.825, Z 387.307, A -116.805, B 80.034, C -131.472, E1 0, E2 0, E3 0, E4 0}
LIN {X 331.791, Y 366.297, Z 385.047, A -116.805, B 80.034, C -131.472, E1 0, E2 0, E3 0, E4 0}
LIN {X 336.773, Y 366.751, Z 384.581, A -116.805, B 80.034, C -131.472, E1 0, E2 0, E3 0, E4 0}
LIN {X 337.066, Y 331.329, Z 390.113, A -116.805, B 80.034, C -131.472, E1 0, E2 0, E3 0, E4 0}
LIN {X 341.996, Y 338.078, Z 388.664, A -116.805, B 80.034, C -131.472, E1 0, E2 0, E3 0, E4 0}
LIN {X 341.752, Y 367.674, Z 384.041, A -116.805, B 80.034, C -131.472, E1 0, E2 0, E3 0, E4 0}
LIN {X 346.73, Y 368.7, Z 383.486, A -116.805, B 80.034, C -131.472, E1 0, E2 0, E3 0, E4 0}
LIN {X 346.931, Y 344.352, Z 387.289, A -116.805, B 80.034, C -131.472, E1 0, E2 0, E3 0, E4 0}
LIN {X 351.852, Y 352.166, Z 385.673, A -116.805, B 80.034, C -131.472, E1 0, E2 0, E3 0, E4 0}
LIN {X 351.71, Y 369.404, Z 382.981, A -116.805, B 80.034, C -131.472, E1 0, E2 0, E3 0, E4 0}
LIN {X 356.69, Y 370.141, Z 382.471, A -116.805, B 80.034, C -131.472, E1 0, E2 0, E3 0, E4 0}
LIN {X 356.775, Y 359.909, Z 384.069, A -116.805, B 80.034, C -131.472, E1 0, E2 0, E3 0, E4 0}
LIN {X 343.779, Y 367.866, Z 383.851, A -116.805, B 80.034, C -131.472, E1 0, E2 0, E3 0, E4 0}
LIN {X 356.603, Y 370.169, Z 382.473, A -116.805, B 80.034, C -131.472, E1 0, E2 0, E3 0, E4 0}
LIN {X 357.297, Y 369.948, Z 382.453, A -116.805, B 80.034, C -131.472, E1 0, E2 0, E3 0, E4 0}
LIN {X 357.327, Y 369.906, Z 382.457, A -116.805, B 80.034, C -131.472, E1 0, E2 0, E3 0, E4 0}
LIN {X 357.895, Y 367.705, Z 382.757, A -116.805, B 80.034, C -131.472, E1 0, E2 0, E3 0, E4 0}
LIN {X 357.854, Y 367.657, Z 382.768, A -116.805, B 80.034, C -131.472, E1 0, E2 0, E3 0, E4 0}
LIN {X 358.546, Y 364.359, Z 383.231, A -116.805, B 80.034, C -131.472, E1 0, E2 0, E3 0, E4 0}
LIN {X 342.444, Y 339.521, Z 388.402, A -116.805, B 80.034, C -131.472, E1 0, E2 0, E3 0, E4 0}
LIN {X 341.986, Y 338.044, Z 388.67, A -116.805, B 80.034, C -131.472, E1 0, E2 0, E3 0, E4 0}
LIN {X 339.402, Y 334.723, Z 389.396, A -116.805, B 80.034, C -131.472, E1 0, E2 0, E3 0, E4 0}
LIN {X 339.025, Y 333.52, Z 389.614, A -116.805, B 80.034, C -131.472, E1 0, E2 0, E3 0, E4 0}
LIN {X 338.256, Y 332.459, Z 389.841, A -116.805, B 80.034, C -131.472, E1 0, E2 0, E3 0, E4 0}
LIN {X 337.441, Y 331.81, Z 390.008, A -116.805, B 80.034, C -131.472, E1 0, E2 0, E3 0, E4 0}
LIN {X 336.347, Y 330.439, Z 390.31, A -116.805, B 80.034, C -131.472, E1 0, E2 0, E3 0, E4 0}
LIN {X 336.066, Y 331.309, Z 390.195, A -116.805, B 80.034, C -131.472, E1 0, E2 0, E3 0, E4 0}
LIN {X 330.19, Y 363.377, Z 385.631, A -116.805, B 80.034, C -131.472, E1 0, E2 0, E3 0, E4 0}
LIN {X 330.593, Y 365.151, Z 385.321, A -116.805, B 80.034, C -131.472, E1 0, E2 0, E3 0, E4 0}
LIN {X 331.82, Y 366.321, Z 385.041, A -116.805, B 80.034, C -131.472, E1 0, E2 0, E3 0, E4 0}
LIN {X 333.258, Y 366.751, Z 384.859, A -116.805, B 80.034, C -131.472, E1 0, E2 0, E3 0, E4 0}
LIN {X 337.314, Y 366.705, Z 384.545, A -116.805, B 80.034, C -131.472, E1 0, E2 0, E3 0, E4 0}
LIN {X 343.779, Y 367.866, Z 383.851, A -116.805, B 80.034, C -131.472, E1 0, E2 0, E3 0, E4 0}
PTP {X 342.707, Y 362.992, Z 432.358, A -116.805, B 80.034, C -131.472, E1 0, E2 0, E3 0, E4 0, S 'B010'}
PTP {A1 5, A2 -90, A3 100, A4 5, A5 -10, A6 -5, E1 0, E2 0, E3 0, E4 0} C_PTP

END
